{attribute 'qualified_only'}
VAR_GLOBAL
	bStart		: BOOL;
	bStop		: BOOL;
	bReset		: BOOL;
	bAuto		: BOOL;
	bManual		: BOOL;
	bFault		: BOOL;
	bSelectAll	: BOOL;
	RNR			: INT;
	bShuttle	: BOOL;
	partID		: STRING;
END_VAR

(* stored: Version 1.1.0.1
   GVL GLOB: Id {22795b31-e4d5-4190-8d90-75899a9009af} *)
